PROGRAM JIG
VAR
END_VAR

END_PROGRAM

(* stored: Version 1.1.0.1, ProductVersion 3.1.4022.18
   POU JIG: Id {17448e34-6352-4909-9200-b00c8ac4245a}, SpecialFunc None *)
